Staubli VAL3: READRECT.pgx

public program readRect(num nHndl_, string x_sCol, num x_nRow, trsf& trOrigin_[], trsf& trSize_[], bool& x_bResult[])
  local bool l_bIsOK
  local bool l_bResult
begin
  // read X coordinate from spreadsheet
  call readNumValue(nHndl_,x_sCol,x_nRow,trOrigin_.x,x_bResult)
  if x_bResult
    // increment column number
    call _incrementCol(x_sCol,l_bIsOK)
    if l_bIsOK
      // read Y coordinate from spreadsheet
      call readNumValue(nHndl_,x_sCol,x_nRow,trOrigin_.y,x_bResult)
      if x_bResult
        // read width from spreadsheet
        call _incrementCol(x_sCol,l_bIsOK)
        if l_bIsOK
          call readNumValue(nHndl_,x_sCol,x_nRow,trSize_.x,x_bResult)
          if x_bResult
            // read height from spreadsheet
            call _incrementCol(x_sCol,l_bIsOK)
            call readNumValue(nHndl_,x_sCol,x_nRow,trSize_.y,x_bResult)
            if x_bResult
              // read RZ from spreadsheet
              call _incrementCol(x_sCol,l_bIsOK)
              if l_bIsOK
                call readNumValue(nHndl_,x_sCol,x_nRow,trOrigin_.rz,x_bResult)
              endIf
            endIf
          endIf
        endIf
      endIf
    endIf
  endIf
end
